(* Logix 5000 project; controller APM_Empacadora Emulate 5570 rev 32.11; software revision 32.00 *)

TASK MainTask (continuous, watchdog 500 ms) : MainProgram

MODULES
   Local : Emulate 5570 (ICP 2, rev 32.11)
END_MODULES

VAR_GLOBAL   (* controller tags *)
   A_Barreras : BOOL;
   A_BrazoCelofan : BOOL;
   A_Caja : BOOL;
   A_ConveyorIngreso : BOOL;
   A_ConveyorSalida : BOOL;
   A_Cuchillas : BOOL;
   A_Freno : BOOL;
   A_Pusher : BOOL;
   BaE : BOOL;
   BaE_Ok : BOOL;
   Bot4 : BOOL;
   Bot4_Ok : BOOL;
   Bot4Al : BOOL;
   Bot4Al_Ok : BOOL;
   BotTunelF : BOOL;
   BotTunelF_Ok : BOOL;
   BotTunelR : BOOL;
   BotTunelR_Ok : BOOL;
   BR : BOOL;
   BR_Ok : BOOL;
   CA_BorrarBotApilado : BOOL;
   CA_BorrarBotIND : BOOL;
   CA_BorrarLinea4Bot : BOOL;
   CA_GenBotApilado : BOOL;
   CA_GenFila4 : BOOL;
   CA_GenPack : BOOL;
   CA_S_BotFila : BOOL;
   CA_S_BotTunel : BOOL;
   Con4Bot : COUNTER := (PRE := 4);
   EnTunel : BOOL;
   EnTunel_Ok : BOOL;
   Etapa0A : BOOL;
   Etapa0E : BOOL;
   Etapa0S : BOOL;
   Etapa1A : BOOL;
   Etapa1E : BOOL;
   Etapa1S : BOOL;
   Etapa2A : BOOL;
   Etapa2E : BOOL;
   Etapa2S : BOOL;
   Etapa3A : BOOL;
   Etapa3E : BOOL;
   Etapa3EA : BOOL;
   Etapa3S : BOOL;
   Etapa4E : BOOL;
   Etapa4EA : BOOL;
   Etapa4S : BOOL;
   Etapa5E : BOOL;
   Etapa5EA : BOOL;
   Etapa5S : BOOL;
   Etapa6E : BOOL;
   Etapa7E : BOOL;
   Etapa7EA : BOOL;
   Etapa8EA : BOOL;
   Etapa9EA : BOOL;
   Fila1 : BOOL;
   Fila1_Ok : BOOL;
   Fila2 : BOOL;
   Fila2_Ok : BOOL;
   Fila3 : BOOL;
   Fila3_Ok : BOOL;
   ND_Start : BOOL;
   ND_Stop : BOOL;
   PosCuchilla : BOOL;
   PosCuchilla_Ok : BOOL;
   S_4BotellaAlineada : BOOL;
   S_BarreraExtendida : BOOL;
   S_BarreraRecogida : BOOL;
   S_BrazoCelofanExtendido : BOOL;
   S_BrazoCelofanRecogido : BOOL;
   S_CajaAbajo : BOOL;
   S_CajaArriba : BOOL;
   S_CuchillasAbiertas : BOOL;
   S_CuchillasCerradas : BOOL;
   S_EntradaBotellas : BOOL;
   S_EntradaTunel : BOOL;
   S_Fila1 : BOOL;
   S_Fila2 : BOOL;
   S_Fila3 : BOOL;
   S_FrenoAbajo : BOOL;
   S_FrenoArriba : BOOL;
   S_IngresoCuchillas : BOOL;
   S_PosCuchillas : BOOL;
   S_PusherRecogido : BOOL;
   S_SalidaCaja : BOOL;
   S_SalidaPackApilado : BOOL;
   S_SalidaTunel : BOOL;
   SalCaja : BOOL;
   SalCaja_Ok : BOOL;
   SalTunel : BOOL;
   SalTunel_Ok : BOOL;
   Sec : BOOL;
   SP : BOOL;
   SP_Ok : BOOL;
   Timer0 : TIMER := (PRE := 6000);
   Timer1 : TIMER := (PRE := 100);
   Timer2 : TIMER := (PRE := 5000);
   Timer3 : TIMER := (PRE := 100);
   Timer4 : TIMER := (PRE := 3000);
   Timer5 : TIMER := (PRE := 3000);
   Timer6 : TIMER := (PRE := 500);
END_VAR

PROGRAM MainProgram   (* main routine MainRoutine *)

ROUTINE MainRoutine   (* ladder *)
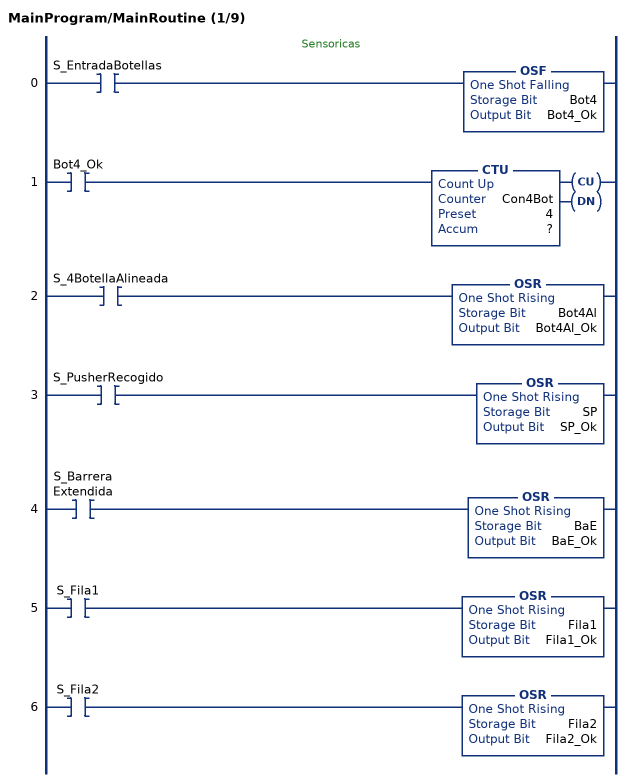
   // Sensoricas
   0: XIC(S_EntradaBotellas)OSF(Bot4,Bot4_Ok);
   1: XIC(Bot4_Ok)CTU(Con4Bot,?,?);
   2: XIC(S_4BotellaAlineada)OSR(Bot4Al,Bot4Al_Ok);
   3: XIC(S_PusherRecogido)OSR(SP,SP_Ok);
   4: XIC(S_BarreraExtendida)OSR(BaE,BaE_Ok);
   5: XIC(S_Fila1)OSR(Fila1,Fila1_Ok);
   6: XIC(S_Fila2)OSR(Fila2,Fila2_Ok);
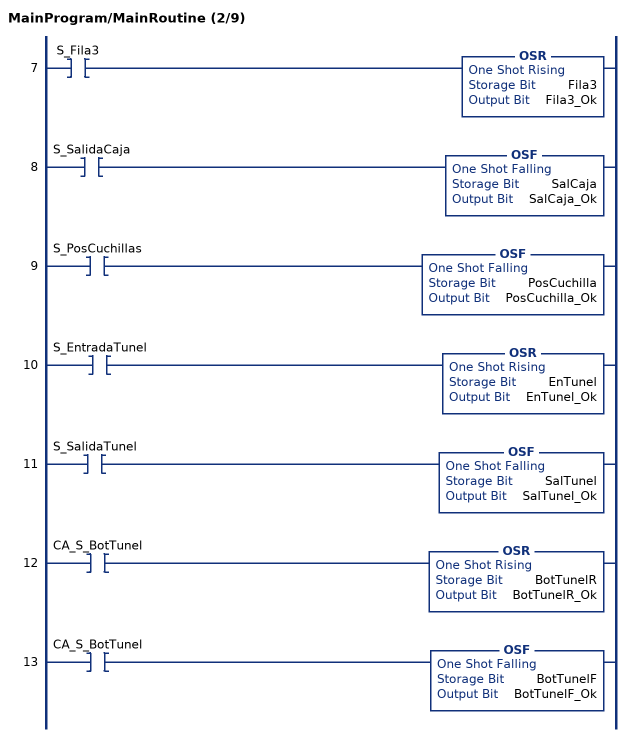
   7: XIC(S_Fila3)OSR(Fila3,Fila3_Ok);
   8: XIC(S_SalidaCaja)OSF(SalCaja,SalCaja_Ok);
   9: XIC(S_PosCuchillas)OSF(PosCuchilla,PosCuchilla_Ok);
   10: XIC(S_EntradaTunel)OSR(EnTunel,EnTunel_Ok);
   11: XIC(S_SalidaTunel)OSF(SalTunel,SalTunel_Ok);
   12: XIC(CA_S_BotTunel)OSR(BotTunelR,BotTunelR_Ok);
   13: XIC(CA_S_BotTunel)OSF(BotTunelF,BotTunelF_Ok);
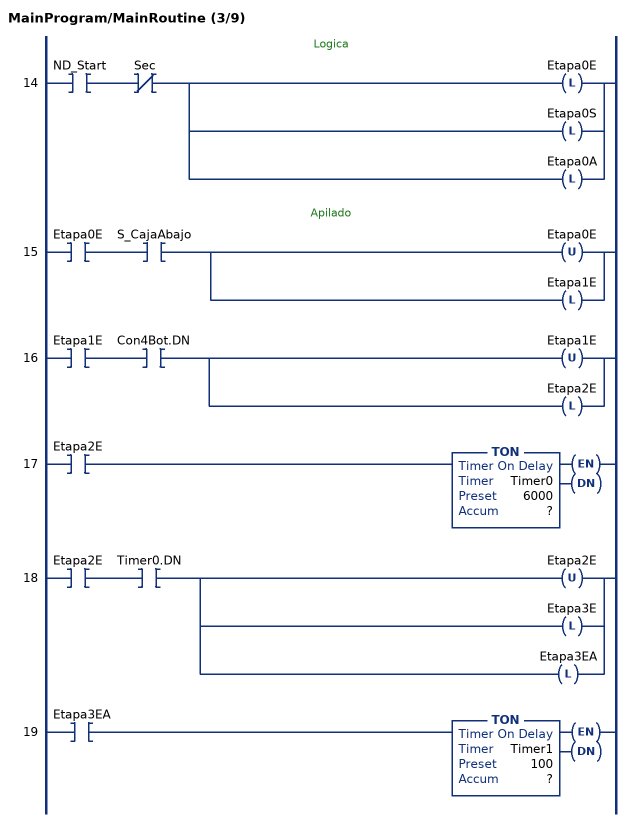
   // Logica
   14: XIC(ND_Start)XIO(Sec)[OTL(Etapa0E) ,[OTL(Etapa0S) ,OTL(Etapa0A) ] ];
   // Apilado
   15: XIC(Etapa0E)XIC(S_CajaAbajo)[OTU(Etapa0E) ,OTL(Etapa1E) ];
   16: XIC(Etapa1E)XIC(Con4Bot.DN)[OTU(Etapa1E) ,OTL(Etapa2E) ];
   17: XIC(Etapa2E)TON(Timer0,?,?);
   18: XIC(Etapa2E)XIC(Timer0.DN)[OTU(Etapa2E) ,[OTL(Etapa3E) ,OTL(Etapa3EA) ] ];
   19: XIC(Etapa3EA)TON(Timer1,?,?);
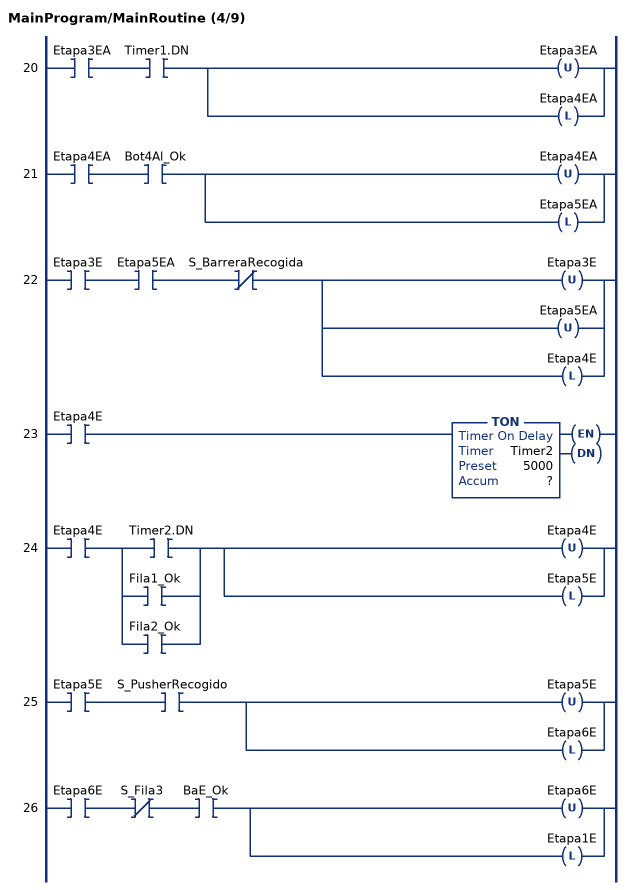
   20: XIC(Etapa3EA)XIC(Timer1.DN)[OTU(Etapa3EA) ,OTL(Etapa4EA) ];
   21: XIC(Etapa4EA)XIC(Bot4Al_Ok)[OTU(Etapa4EA) ,OTL(Etapa5EA) ];
   22: XIC(Etapa3E)XIC(Etapa5EA)XIO(S_BarreraRecogida)[OTU(Etapa3E) ,[OTU(Etapa5EA) ,OTL(Etapa4E) ] ];
   23: XIC(Etapa4E)TON(Timer2,?,?);
   24: XIC(Etapa4E)[XIC(Timer2.DN) ,[XIC(Fila1_Ok) ,XIC(Fila2_Ok) ] ][OTU(Etapa4E) ,OTL(Etapa5E) ];
   25: XIC(Etapa5E)XIC(S_PusherRecogido)[OTU(Etapa5E) ,OTL(Etapa6E) ];
   26: XIC(Etapa6E)XIO(S_Fila3)XIC(BaE_Ok)[OTU(Etapa6E) ,OTL(Etapa1E) ];
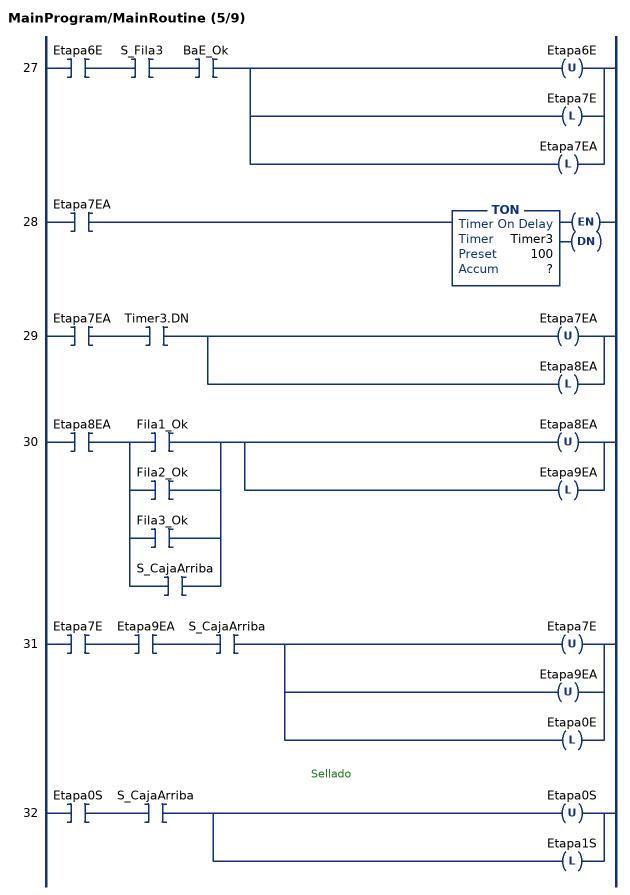
   27: XIC(Etapa6E)XIC(S_Fila3)XIC(BaE_Ok)[OTU(Etapa6E) ,[OTL(Etapa7E) ,OTL(Etapa7EA) ] ];
   28: XIC(Etapa7EA)TON(Timer3,?,?);
   29: XIC(Etapa7EA)XIC(Timer3.DN)[OTU(Etapa7EA) ,OTL(Etapa8EA) ];
   30: XIC(Etapa8EA)[XIC(Fila1_Ok) ,[XIC(Fila2_Ok) ,[XIC(Fila3_Ok) ,XIC(S_CajaArriba) ] ] ][OTU(Etapa8EA) ,OTL(Etapa9EA) ];
   31: XIC(Etapa7E)XIC(Etapa9EA)XIC(S_CajaArriba)[OTU(Etapa7E) ,[OTU(Etapa9EA) ,OTL(Etapa0E) ] ];
   // Sellado
   32: XIC(Etapa0S)XIC(S_CajaArriba)[OTU(Etapa0S) ,OTL(Etapa1S) ];
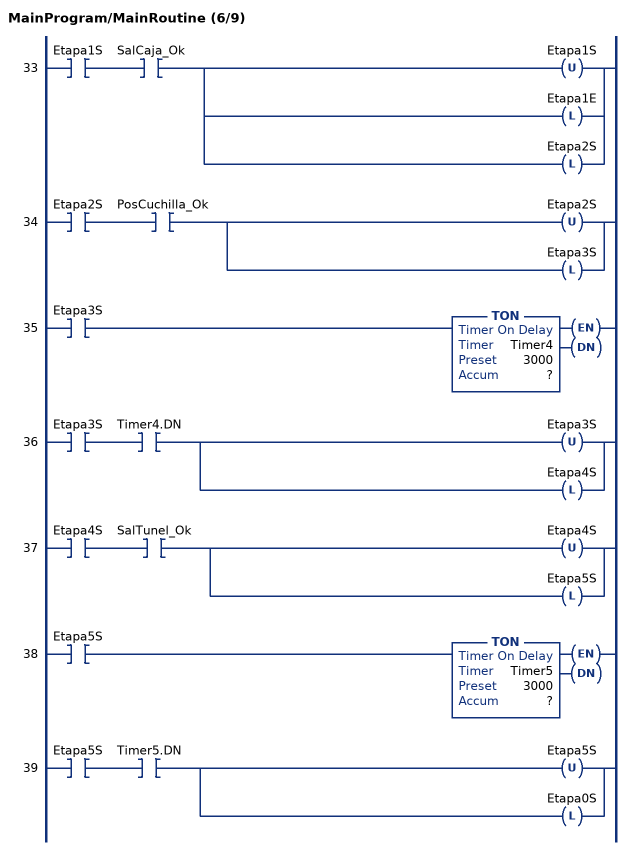
   33: XIC(Etapa1S)XIC(SalCaja_Ok)[OTU(Etapa1S) ,[OTL(Etapa1E) ,OTL(Etapa2S) ] ];
   34: XIC(Etapa2S)XIC(PosCuchilla_Ok)[OTU(Etapa2S) ,OTL(Etapa3S) ];
   35: XIC(Etapa3S)TON(Timer4,?,?);
   36: XIC(Etapa3S)XIC(Timer4.DN)[OTU(Etapa3S) ,OTL(Etapa4S) ];
   37: XIC(Etapa4S)XIC(SalTunel_Ok)[OTU(Etapa4S) ,OTL(Etapa5S) ];
   38: XIC(Etapa5S)TON(Timer5,?,?);
   39: XIC(Etapa5S)XIC(Timer5.DN)[OTU(Etapa5S) ,OTL(Etapa0S) ];
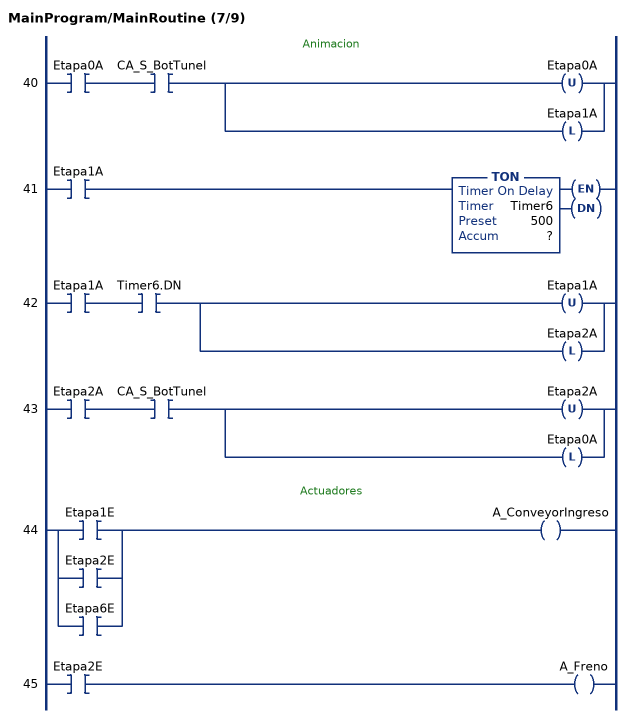
   // Animacion
   40: XIC(Etapa0A)XIC(CA_S_BotTunel)[OTU(Etapa0A) ,OTL(Etapa1A) ];
   41: XIC(Etapa1A)TON(Timer6,?,?);
   42: XIC(Etapa1A)XIC(Timer6.DN)[OTU(Etapa1A) ,OTL(Etapa2A) ];
   43: XIC(Etapa2A)XIC(CA_S_BotTunel)[OTU(Etapa2A) ,OTL(Etapa0A) ];
   // Actuadores
   44: [XIC(Etapa1E) ,[XIC(Etapa2E) ,XIC(Etapa6E) ] ]OTE(A_ConveyorIngreso);
   45: XIC(Etapa2E)OTE(A_Freno);
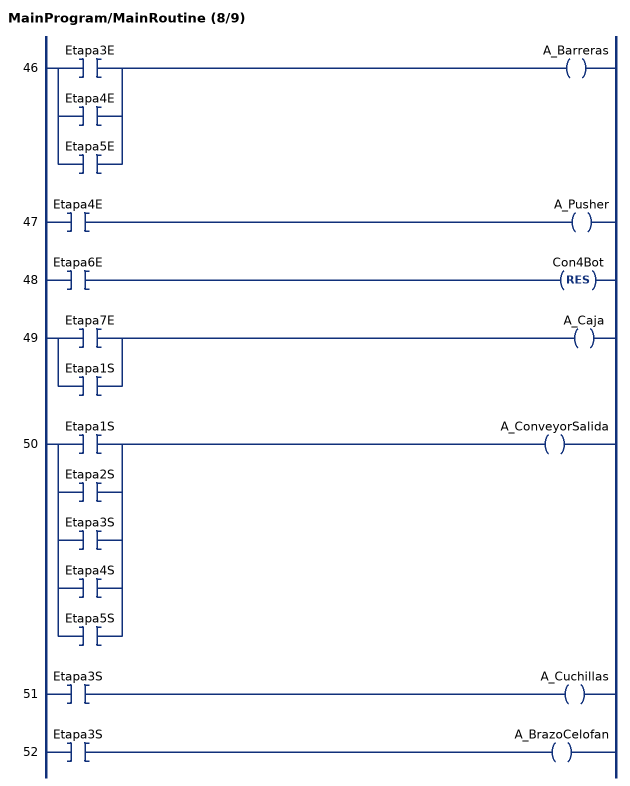
   46: [XIC(Etapa3E) ,[XIC(Etapa4E) ,XIC(Etapa5E) ] ]OTE(A_Barreras);
   47: XIC(Etapa4E)OTE(A_Pusher);
   48: XIC(Etapa6E)RES(Con4Bot);
   49: [XIC(Etapa7E) ,XIC(Etapa1S) ]OTE(A_Caja);
   50: [XIC(Etapa1S) ,[XIC(Etapa2S) ,[XIC(Etapa3S) ,[XIC(Etapa4S) ,XIC(Etapa5S) ] ] ] ]OTE(A_ConveyorSalida);
   51: XIC(Etapa3S)OTE(A_Cuchillas);
   52: XIC(Etapa3S)OTE(A_BrazoCelofan);
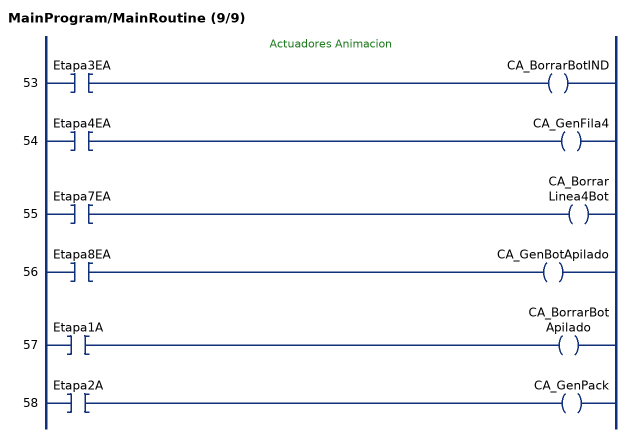
   // Actuadores Animacion
   53: XIC(Etapa3EA)OTE(CA_BorrarBotIND);
   54: XIC(Etapa4EA)OTE(CA_GenFila4);
   55: XIC(Etapa7EA)OTE(CA_BorrarLinea4Bot);
   56: XIC(Etapa8EA)OTE(CA_GenBotApilado);
   57: XIC(Etapa1A)OTE(CA_BorrarBotApilado);
   58: XIC(Etapa2A)OTE(CA_GenPack);
END_ROUTINE
END_PROGRAM
